{attribute 'no_check'}
//Cylinder with runtime status, extended from FB Cylinder
FUNCTION_BLOCK CylinderExt EXTENDS Cylinder 
VAR_OUTPUT CONSTANT
END_VAR
VAR_INPUT  

END_VAR                                     			
VAR_OUTPUT     			
	RuntimeWP												:	TIME;
	RuntimeBP												:	TIME;
END_VAR
VAR
END_VAR

	(* Cylinder	with runtime status 												*)
	(********************************************************************************)

(* Call super ********************************************************)
	SUPER^();
	
(*********************************************************************)

METHOD PROTECTED _runtimeChk : BOOL
VAR_INPUT
END_VAR
VAR
	memRtBP												:	TIME;
	memRtWP												:	TIME;
END_VAR
(* Record current runtime **********************************************)
	memRtBP													:= tonErrBasePos.ET;
	memRtWP													:= TonErrWorkPos.ET;
	
(* Call time *********************************************************)
	SUPER^._runtimeChk();
	
(* Record last runtime *********************************************)
	IF memRtWP > T#0MS AND NOT tonErrWorkPos.IN AND NOT tonErrWorkPos.Q
	THEN
		RuntimeWP											:= memRtWP;
	END_IF
	
	IF memRtBP > T#0MS AND NOT tonErrBasePos.IN AND NOT tonErrBasePos.Q
	THEN
		RuntimeBP											:= memRtBP;
	END_IF
					
(*********************************************************************)
	_runtimeChk												:= TRUE;

(**********************************************************************)
END_METHOD

END_FUNCTION_BLOCK

(* stored: Version 1.1.0.1, ProductVersion 3.1.4024.6
   POU CylinderExt: Id {2b722628-ffee-4ec8-9c64-bdd463427979}, SpecialFunc None
   Method _runtimeChk: Id {548c6c7d-1913-470d-ae27-f4e9c92353ee} *)
